ABB RobotStudio station: TrabalhoN2_20220517-152928.rsstn

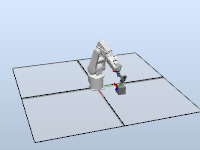
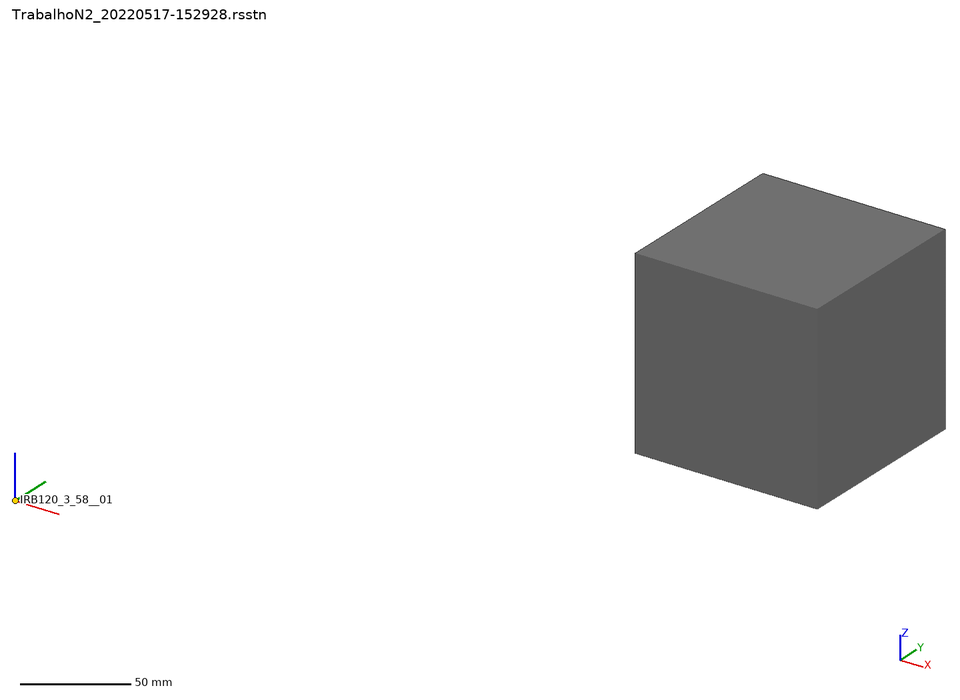
[picture v1: parts stored in the station drawn from their meshes, with robot base, taught points and paths (robot models come from the ABB library and are not in the file)]
Station TrabalhoN2 (saved by RobotStudio 22.1.9826.0)
Controller IRB120_3_58
  mechanical unit ROB_1: IRB120_3_58__01, 6 joints, base frame (0, 0, 0) mm
Layout (positions relative to the parent item):
  - IRB120_3_58__01 [mechanism, from Robots\IRB120_3_58_G_01.rslib] at (0, 0, 0) mm; joint values [0.4501, 0.292, 0.3542, 0.2036, 0.8516, -0.3356] (rad or m)
  - caixa [part] at (100, 100, 0) mm, size 100 x 100 x 100 mm
  - MyTool [mechanism, from Training Objects\myTool.rslib] at (325.6, 169.49, 351.68) mm, rotated rx 172.37 ry 6.42 rz -142.79 deg
  - Positioner [smart component, from Components\Positioner.rslib]
      properties: Object=caixa; Position=[0.1 0.1 0]; Orientation=[0 0 0]; Reference=Global; ReferenceObject=(none)
  - Detacher [smart component, from Components\Detacher.rslib]
      properties: Child=caixa; KeepPosition=true
  - Attacher [smart component, from Components\Attacher.rslib]
      properties: Parent=MyTool; Flange=0; Child=caixa; Mount=false; Offset=[0 0 0]; Orientation=[0 0 0]
Attachment: MyTool is attached to IRB120_3_58__01 / Link6
Station signals: DI Digital1
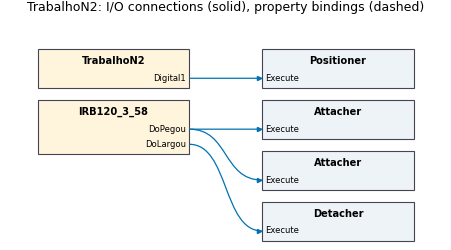
Station logic (signal -> signal, property => property):
  TrabalhoN2.Digital1 -> Positioner.Execute
  IRB120_3_58.DoPegou -> Attacher.Execute
  IRB120_3_58.DoLargou -> Detacher.Execute
  IRB120_3_58.DoPegou -> Attacher.Execute
Targets, tools, work objects and paths stored in the station, written as RAPID:
! task T_ROB1
MODULE CalibData
  PERS tooldata MyTool:=[TRUE,[[31.792631019,0,229.638935148],[0.945518576,0,0.325568154,0]],[1,[0,0,1],[1,0,0,0],0,0,0]];
ENDMODULE

